Staubli VAL3: N11_Banyera.pgx

program N11_Banyera()
  local pointRx l_pBanyera
begin

  // Anar al punt de la banyera
  l_pBanyera=pBanyera[aioGet(aiNumBanyera)]
  l_pBanyera.trsf.x=l_pBanyera.trsf.x+nXOffset
  l_pBanyera.trsf.y=l_pBanyera.trsf.y+nYOffset
  l_pBanyera.trsf.z=l_pBanyera.trsf.z+nZOffset
  movel(l_pBanyera,tToolActiva,mLent)
  waitEndMove()

  bTaskDone=true
end
